FUNCTION_BLOCK offline_fb
VAR
	cylinder_1: cylinder_2_pos;
	cylinder_2: cylinder_2_pos;
	cylinder_3: cylinder_2_pos;
	cylinder_4: cylinder_2_pos;
	cylinder_5: cylinder_2_pos;
	cylinder_6: cylinder_2_pos;
	cylinder_7: cylinder_2_pos;
	cylinder_8: cylinder_2_pos;
	cylinder_9: cylinder_2_pos;
	cylinder_10: cylinder_2_pos;
	servo_1: servo;
	servo_2: servo;
	servo_3: servo;
	servo_4: servo;
	servo_5: servo;
	servo_6: servo;
	servo_7: servo;
	servo_8: servo;
	servo_9: servo;
	servo_10: servo;
END_VAR

VAR_OUTPUT
	
	// cylinder out
	
cyl_work_fb_1   :BOOL;
cyl_home_fb_1   :BOOL;
cyl_work_fb_2   :BOOL;
cyl_home_fb_2   :BOOL;
cyl_work_fb_3   :BOOL;
cyl_home_fb_3   :BOOL;
cyl_work_fb_4   :BOOL;
cyl_home_fb_4   :BOOL;
cyl_work_fb_5   :BOOL;
cyl_home_fb_5   :BOOL;
cyl_work_fb_6   :BOOL;
cyl_home_fb_6   :BOOL;
cyl_work_fb_7   :BOOL;
cyl_home_fb_7   :BOOL;
cyl_work_fb_8   :BOOL;
cyl_home_fb_8   :BOOL;
cyl_work_fb_9   :BOOL;
cyl_home_fb_9   :BOOL;
cyl_work_fb_10  :BOOL;
cyl_home_fb_10  :BOOL;

// servo out

Actual_position_1       :real;
Actual_position_2       :real;
Actual_position_3       :real;
Actual_position_4       :real;
Actual_position_5       :real;
Actual_position_6       :real;
Actual_position_7       :real;
Actual_position_8       :real;
Actual_position_9       :real;
Actual_position_10      :real;

END_VAR
VAR_INPUT 
	
	//general
	offline_test      :BOOL;
	error_bit         :BOOL;
	
	// cylinder input set

cyl_work_sol_1        :BOOL;
cyl_home_sol_1        :BOOL;
delay_1_1             :LTIME;
delay_2_1             :LTIME;

cyl_work_sol_2        :BOOL;
cyl_home_sol_2        :BOOL;
delay_1_2             :LTIME;
delay_2_2             :LTIME;

cyl_work_sol_3        :BOOL;
cyl_home_sol_3        :BOOL;
delay_1_3             :LTIME;
delay_2_3             :LTIME;

cyl_work_sol_4        :BOOL;
cyl_home_sol_4        :BOOL;
delay_1_4             :LTIME;
delay_2_4             :LTIME;

cyl_work_sol_5        :BOOL;
cyl_home_sol_5        :BOOL;
delay_1_5             :LTIME;
delay_2_5             :LTIME;

cyl_work_sol_6        :BOOL;
cyl_home_sol_6        :BOOL;
delay_1_6             :LTIME;
delay_2_6             :LTIME;

cyl_work_sol_7        :BOOL;
cyl_home_sol_7        :BOOL;
delay_1_7             :LTIME;
delay_2_7             :LTIME;

cyl_work_sol_8        :BOOL;
cyl_home_sol_8        :BOOL;
delay_1_8             :LTIME;
delay_2_8             :LTIME;

cyl_work_sol_9        :BOOL;
cyl_home_sol_9        :BOOL;
delay_1_9             :LTIME;
delay_2_9             :LTIME;

cyl_work_sol_10       :bool;
cyl_home_sol_10       :BOOL;
delay_1_10            :LTIME;
delay_2_10            :LTIME;  
  
// servo input set

servo_absolute_1        :BOOL;
target_position_1       :REAL;
s_delay_1_1             :LTIME;

servo_absolute_2        :BOOL;
target_position_2       :REAL;
s_delay_1_2             :LTIME;

servo_absolute_3        :BOOL;
target_position_3       :REAL;
s_delay_1_3             :LTIME;

servo_absolute_4        :BOOL;
target_position_4       :REAL;
s_delay_1_4             :LTIME;

servo_absolute_5        :BOOL;
target_position_5       :REAL;
s_delay_1_5             :LTIME;

servo_absolute_6        :BOOL;
target_position_6       :REAL;
s_delay_1_6             :LTIME;

servo_absolute_7        :BOOL;
target_position_7       :REAL;
s_delay_1_7             :LTIME;

servo_absolute_8        :BOOL;
target_position_8       :REAL;
s_delay_1_8             :LTIME;

servo_absolute_9        :BOOL;
target_position_9       :REAL;
s_delay_1_9             :LTIME;

servo_absolute_10       :BOOL;
target_position_10      :REAL;
s_delay_1_10            :LTIME;

END_VAR

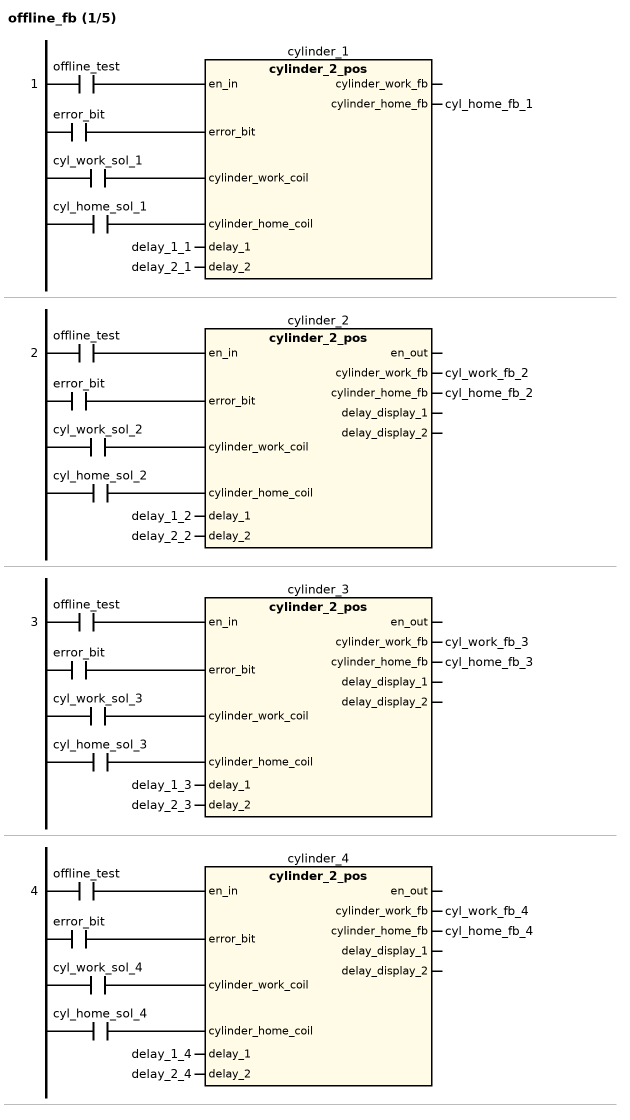
// NETWORK 1
cylinder_1(
    en_in := offline_test,
    error_bit := error_bit,
    cylinder_work_coil := cyl_work_sol_1,
    cylinder_home_coil := cyl_home_sol_1,
    delay_1 := delay_1_1,
    delay_2 := delay_2_1,
    cylinder_home_fb => cyl_home_fb_1); // cylinder_2_pos

// NETWORK 2
cylinder_2(
    en_in := offline_test,
    error_bit := error_bit,
    cylinder_work_coil := cyl_work_sol_2,
    cylinder_home_coil := cyl_home_sol_2,
    delay_1 := delay_1_2,
    delay_2 := delay_2_2,
    cylinder_work_fb => cyl_work_fb_2,
    cylinder_home_fb => cyl_home_fb_2); // cylinder_2_pos

// NETWORK 3
cylinder_3(
    en_in := offline_test,
    error_bit := error_bit,
    cylinder_work_coil := cyl_work_sol_3,
    cylinder_home_coil := cyl_home_sol_3,
    delay_1 := delay_1_3,
    delay_2 := delay_2_3,
    cylinder_work_fb => cyl_work_fb_3,
    cylinder_home_fb => cyl_home_fb_3); // cylinder_2_pos

// NETWORK 4
cylinder_4(
    en_in := offline_test,
    error_bit := error_bit,
    cylinder_work_coil := cyl_work_sol_4,
    cylinder_home_coil := cyl_home_sol_4,
    delay_1 := delay_1_4,
    delay_2 := delay_2_4,
    cylinder_work_fb => cyl_work_fb_4,
    cylinder_home_fb => cyl_home_fb_4); // cylinder_2_pos

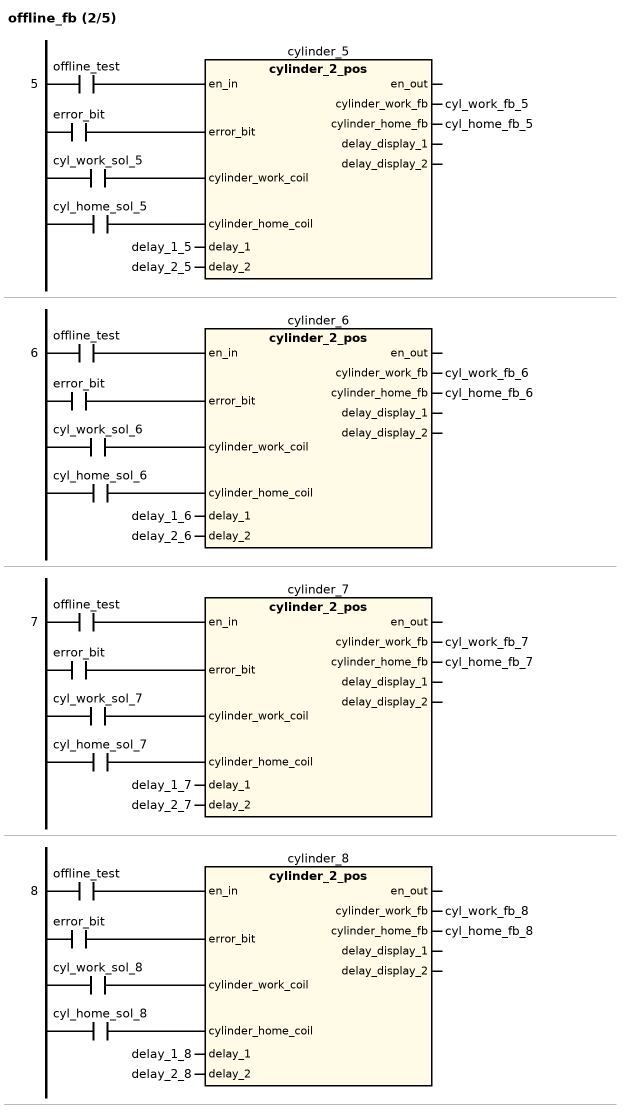
// NETWORK 5
cylinder_5(
    en_in := offline_test,
    error_bit := error_bit,
    cylinder_work_coil := cyl_work_sol_5,
    cylinder_home_coil := cyl_home_sol_5,
    delay_1 := delay_1_5,
    delay_2 := delay_2_5,
    cylinder_work_fb => cyl_work_fb_5,
    cylinder_home_fb => cyl_home_fb_5); // cylinder_2_pos

// NETWORK 6
cylinder_6(
    en_in := offline_test,
    error_bit := error_bit,
    cylinder_work_coil := cyl_work_sol_6,
    cylinder_home_coil := cyl_home_sol_6,
    delay_1 := delay_1_6,
    delay_2 := delay_2_6,
    cylinder_work_fb => cyl_work_fb_6,
    cylinder_home_fb => cyl_home_fb_6); // cylinder_2_pos

// NETWORK 7
cylinder_7(
    en_in := offline_test,
    error_bit := error_bit,
    cylinder_work_coil := cyl_work_sol_7,
    cylinder_home_coil := cyl_home_sol_7,
    delay_1 := delay_1_7,
    delay_2 := delay_2_7,
    cylinder_work_fb => cyl_work_fb_7,
    cylinder_home_fb => cyl_home_fb_7); // cylinder_2_pos

// NETWORK 8
cylinder_8(
    en_in := offline_test,
    error_bit := error_bit,
    cylinder_work_coil := cyl_work_sol_8,
    cylinder_home_coil := cyl_home_sol_8,
    delay_1 := delay_1_8,
    delay_2 := delay_2_8,
    cylinder_work_fb => cyl_work_fb_8,
    cylinder_home_fb => cyl_home_fb_8); // cylinder_2_pos

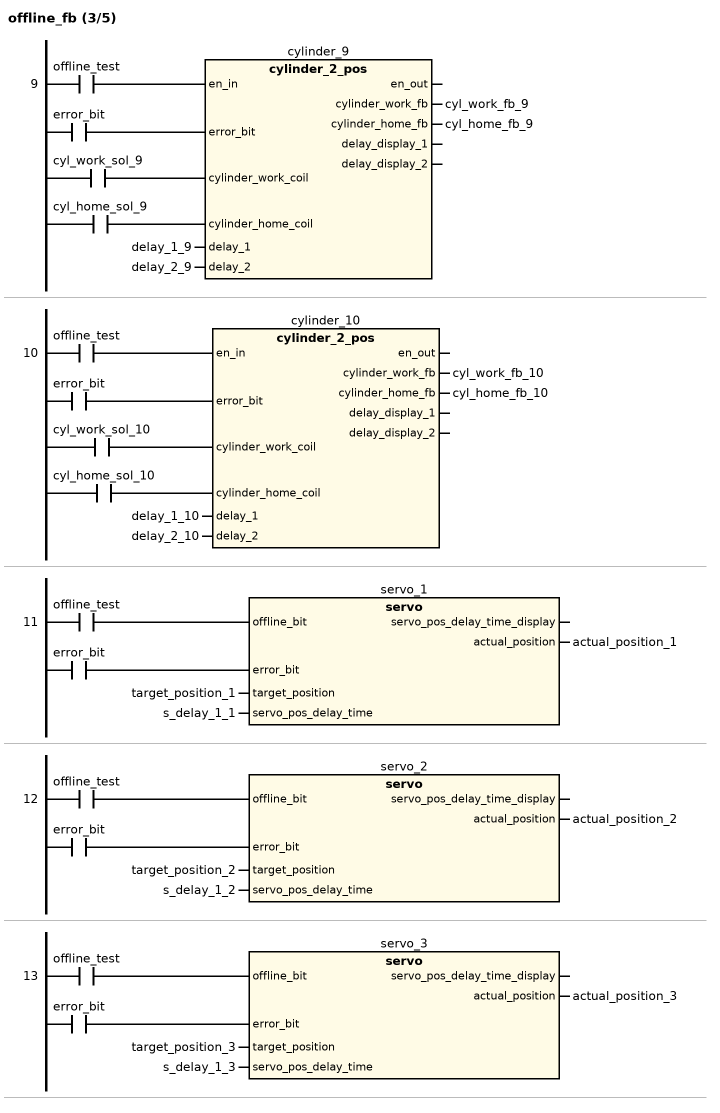
// NETWORK 9
cylinder_9(
    en_in := offline_test,
    error_bit := error_bit,
    cylinder_work_coil := cyl_work_sol_9,
    cylinder_home_coil := cyl_home_sol_9,
    delay_1 := delay_1_9,
    delay_2 := delay_2_9,
    cylinder_work_fb => cyl_work_fb_9,
    cylinder_home_fb => cyl_home_fb_9); // cylinder_2_pos

// NETWORK 10
cylinder_10(
    en_in := offline_test,
    error_bit := error_bit,
    cylinder_work_coil := cyl_work_sol_10,
    cylinder_home_coil := cyl_home_sol_10,
    delay_1 := delay_1_10,
    delay_2 := delay_2_10,
    cylinder_work_fb => cyl_work_fb_10,
    cylinder_home_fb => cyl_home_fb_10); // cylinder_2_pos

// NETWORK 11
servo_1(
    offline_bit := offline_test,
    error_bit := error_bit,
    target_position := target_position_1,
    servo_pos_delay_time := s_delay_1_1,
    actual_position => actual_position_1); // servo

// NETWORK 12
servo_2(
    offline_bit := offline_test,
    error_bit := error_bit,
    target_position := target_position_2,
    servo_pos_delay_time := s_delay_1_2,
    actual_position => actual_position_2); // servo

// NETWORK 13
servo_3(
    offline_bit := offline_test,
    error_bit := error_bit,
    target_position := target_position_3,
    servo_pos_delay_time := s_delay_1_3,
    actual_position => actual_position_3); // servo

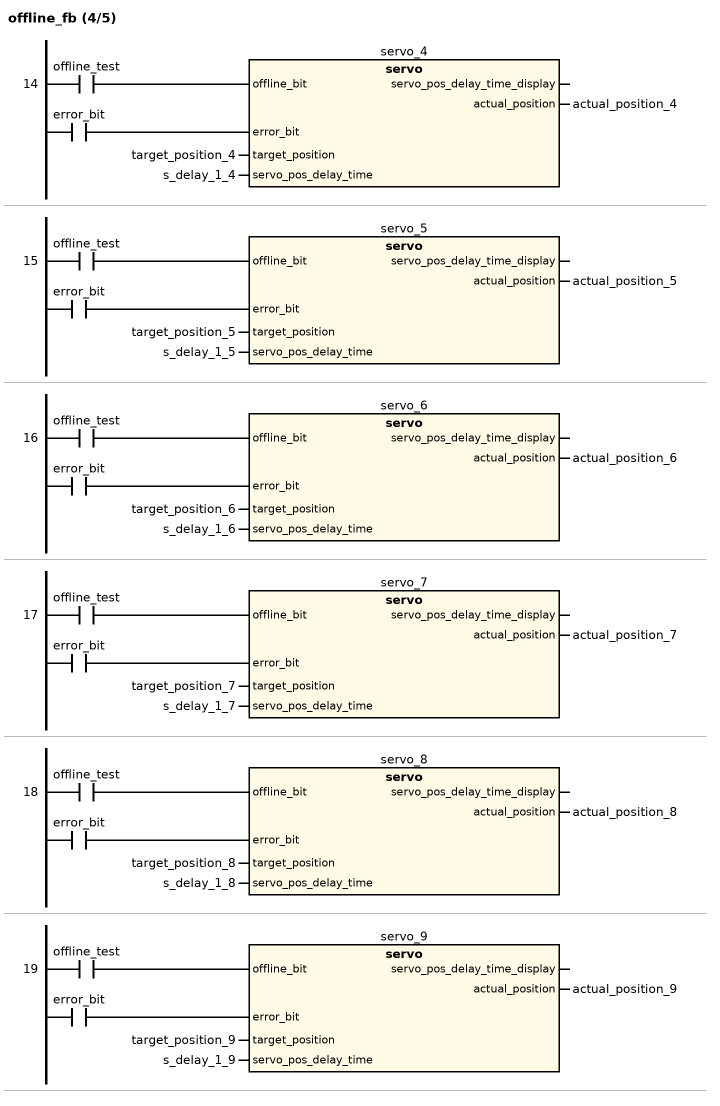
// NETWORK 14
servo_4(
    offline_bit := offline_test,
    error_bit := error_bit,
    target_position := target_position_4,
    servo_pos_delay_time := s_delay_1_4,
    actual_position => actual_position_4); // servo

// NETWORK 15
servo_5(
    offline_bit := offline_test,
    error_bit := error_bit,
    target_position := target_position_5,
    servo_pos_delay_time := s_delay_1_5,
    actual_position => actual_position_5); // servo

// NETWORK 16
servo_6(
    offline_bit := offline_test,
    error_bit := error_bit,
    target_position := target_position_6,
    servo_pos_delay_time := s_delay_1_6,
    actual_position => actual_position_6); // servo

// NETWORK 17
servo_7(
    offline_bit := offline_test,
    error_bit := error_bit,
    target_position := target_position_7,
    servo_pos_delay_time := s_delay_1_7,
    actual_position => actual_position_7); // servo

// NETWORK 18
servo_8(
    offline_bit := offline_test,
    error_bit := error_bit,
    target_position := target_position_8,
    servo_pos_delay_time := s_delay_1_8,
    actual_position => actual_position_8); // servo

// NETWORK 19
servo_9(
    offline_bit := offline_test,
    error_bit := error_bit,
    target_position := target_position_9,
    servo_pos_delay_time := s_delay_1_9,
    actual_position => actual_position_9); // servo

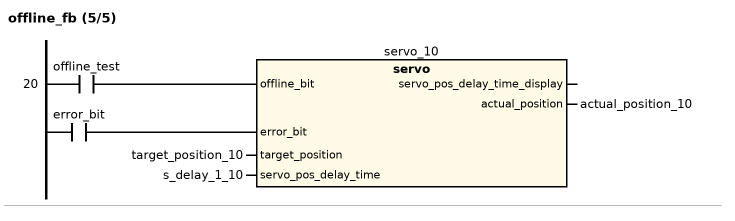
// NETWORK 20
servo_10(
    offline_bit := offline_test,
    error_bit := error_bit,
    target_position := target_position_10,
    servo_pos_delay_time := s_delay_1_10,
    actual_position => actual_position_10); // servo

END_FUNCTION_BLOCK

(* stored: Version 1.1.0.1, ProductVersion 3.1.4024.11
   POU offline_fb: Id {f27bf9ac-8c25-44bd-a8ce-4c396fb6cfd0}, SpecialFunc None *)
